Yaskawa INFORM job: SHIP.JBI

/JOB
//NAME SHIP
//POS
///NPOS 1,0,0,0,0,0
///TOOL 0
///POSTYPE PULSE
///PULSE
C00000=2,-173489,-159173,90424,-90135,10
//INST
///DATE 2021/09/20 14:20
///ATTR SC,RW
///GROUP1 RB1
NOP
MOVJ C00000 VJ=10.00
END
